// TIA Portal V17 export
// export: Created 2023-12-22T15:03:09.2394525Z, ExportSetting WithDefaults, DisplayName Totally Integrated Automation Portal, DisplayVersion V17, DisplayName TIA Portal Openness, DisplayVersion V17, DisplayName TIA Portal Version Control Interface, DisplayVersion V17, DisplayName STEP 7 Professional, DisplayVersion V17, DisplayName STEP 7 Safety, DisplayVersion V17, DisplayName WinCC Advanced, DisplayVersion V17
DATA_BLOCK "AUMA_KP_4_DB"   // DB424
{ S7_Optimized_Access := 'FALSE' }
VERSION : 0.1
// stored: AutoNumber false, DBAccessibleFromOPCUA true, DBAccessibleFromWebserver true, IsOnlyStoredInLoadMemory false, IsWriteProtectedInAS false
   VAR RETAIN
      AUMA : Array[0..10] of Struct   // Чтение - Input Register (04), Запись - Holding Register (06)
         Message : Struct   // Сообщения
            Open : Bool;   // - конечное положение ОТКРЫТО
            Close : Bool;   // - конечное положение ЗАКРЫТО
            Pos_Ok : Bool;   // - положение уставки достигнуто
            NotReady : Bool;   // - не готов ДИСТ.
            Opening : Bool;   // - работет ОТКРЫТИЕ
            Closing : Bool;   // - работает ЗАКРЫТИЕ
            Warning : Bool;   // - предупреждения
            Error : Bool;   // - ошибки
            Err_Termo : Bool;   // - термическая ошибка
            Err_Power : Bool;   // - сбой фазы
            Sel_Dist : Bool;   // - селектор ДИСТ
            Sel_Local : Bool;   // - селектор МЕСТНЫЙ
            FB_Open : Bool;   // - концевик ОТКРЫТО
            FB_Close : Bool;   // - концевик ЗАКРЫТО
            Err_Open : Bool;   // - момент выключения ОТКРЫТО
            Err_Close : Bool;   // - момент выключения ЗАКРЫТО
         END_STRUCT;
         Position : Int;   // Фактическое положение
         Device : Struct   // Статус
            NotReady_Dist : Bool;   // - не готов ДИСТ
            Warning : Bool;   // - предупреждние
            Alarm : Bool;   // - сбой
            Req_Service : Bool;   // - требуется тех обслуживание
            NonSpec : Bool;   // - вне спецификации
            Check : Bool;   // - проверка функций
            Error : Bool;   // - сбой
            Normal : Bool;   // - устройство в норме
            Pos_Pause : Bool;   // - активна пауза в перемещении
            Pos_Any : Bool;   // - в промежуточном положение
            Pos_Section : Bool;   // - достигнут участок пошагового режима
            Pos_Ok : Bool;   // - достигнута позиция MPV
            Busy : Bool;   // - привод работает
            Hand : Bool;   // - перемещение с помощью маховика
            Dist : Bool;   // - перемещение в дистанционном режиме
            Local : Bool;   // - перемещение в местном режиме
         END_STRUCT;
         addr_1003 : Word;
         CMD_last : Struct   // Управление
            Open : Bool;
            Close : Bool;
            SetPoint : Bool;
            Reset : Bool;
            Stop : Bool;
            res_0 : Bool;
            res_1 : Bool;
            res_2 : Bool;
            sp_0 : Bool;
            sp_1 : Bool;
            sp_2 : Bool;
            sp_3 : Bool;
            sp_4 : Bool;
            sp_5 : Bool;
            sp_6 : Bool;
            sp_7 : Bool;
            Position : Int;
            xLocalON : Bool;
            xUnLock_Open : Bool;
            xUnLock_Close : Bool;
            xBtON : Bool;
            xCh1 : Bool;
            xCh2 : Bool;
            xAlarm : Bool;
            PVST : Bool;
            res_00 : Bool;
            res_01 : Bool;
            res_02 : Bool;
            res_03 : Bool;
            res_04 : Bool;
            res_05 : Bool;
            res_06 : Bool;
            res_07 : Bool;
         END_STRUCT;
         CMD : Struct   // Управление
            Open : Bool;
            Close : Bool;
            SetPoint : Bool;
            Reset : Bool;
            Stop : Bool;
            res_0 : Bool;
            res_1 : Bool;
            res_2 : Bool;
            sp_0 : Bool;
            sp_1 : Bool;
            sp_2 : Bool;
            sp_3 : Bool;
            sp_4 : Bool;
            sp_5 : Bool;
            sp_6 : Bool;
            sp_7 : Bool;
            Position : Int;
            xLocalON : Bool;
            xUnLock_Open : Bool;
            xUnLock_Close : Bool;
            xBtON : Bool;
            xCh1 : Bool;
            xCh2 : Bool;
            xAlarm : Bool;
            PVST : Bool;
            res_00 : Bool;
            res_01 : Bool;
            res_02 : Bool;
            res_03 : Bool;
            res_04 : Bool;
            res_05 : Bool;
            res_06 : Bool;
            res_07 : Bool;
         END_STRUCT;
         Use { S7_SetPoint := 'True'} : Bool;
         Link : Bool;
         NoRead : Bool;
         NoWrite : Bool;
         Update : Bool;
         ID { S7_SetPoint := 'True'} : Int;
         ADDR { S7_SetPoint := 'True'} : UInt;
         Speed : Byte;
         "Name" { S7_SetPoint := 'True'} : String[10];
      END_STRUCT;
   END_VAR
BEGIN
   AUMA[0].CMD_last.sp_2 := TRUE;
   AUMA[0].CMD_last.sp_5 := TRUE;
   AUMA[0].CMD_last.sp_6 := TRUE;
   AUMA[0].CMD.sp_2 := TRUE;
   AUMA[0].CMD.sp_5 := TRUE;
   AUMA[0].CMD.sp_6 := TRUE;
   AUMA[0].Use := FALSE;
   AUMA[1..5].Use := TRUE;
   AUMA[6..10].Use := FALSE;
   AUMA[0].ID := 0;
   AUMA[1..5].ID := 12;
   AUMA[6..9].ID := 2;
   AUMA[10].ID := 0;
   AUMA[0..1].ADDR := 21;
   AUMA[2].ADDR := 22;
   AUMA[3].ADDR := 23;
   AUMA[4].ADDR := 24;
   AUMA[5].ADDR := 25;
   AUMA[6..10].ADDR := 0;
   AUMA[0]."Name" := 'M136';
   AUMA[1]."Name" := 'M205';
   AUMA[2]."Name" := 'M204';
   AUMA[3]."Name" := 'M202';
   AUMA[4]."Name" := 'M203';
   AUMA[5]."Name" := 'K201';
   AUMA[6..10]."Name" := '';
END_DATA_BLOCK
